// TwinCAT 3 PLC project SeedraPLC
// ProgramVersion: 3.1.4023.0
// libraries:
//   SPT Base Types, * (Beckhoff Automation LLC)
//   SPT Components, * (Beckhoff Automation LLC)
//   SPT Event Logger, * (Beckhoff Automation LLC)
//   SPT Motion Control, * (Beckhoff Automation LLC)
//   SPT Utilities, * (Beckhoff Automation LLC)
//   Tc2_EtherCAT, * (Beckhoff Automation GmbH)
//   Tc2_MC2, * (Beckhoff Automation GmbH)
//   Tc2_Standard, * (Beckhoff Automation GmbH)
//   Tc2_System, * (Beckhoff Automation GmbH)
//   Tc3_EventLogger, * (Beckhoff Automation GmbH)
//   Tc3_Module, * (Beckhoff Automation GmbH)
//   Tc3_PackML_V2, * (Beckhoff Automation GmbH)
//   VisuDialogs, * (System)
//   VisuSymbols,newest,System
// project tree:
//   / GlobalTextList.TcGTLO, MAIN.TcPOU, TaskPLC.TcTTO, VisualizationManager.TcVMO (not stored)
//   GVL/ IO.TcGVL, SafetyGlobalVariableList.TcGVL
//   Machine/Components/ FB_GantryXYCylinder.TcPOU, I_Cylinder.TcIO (not stored), ST_CylinderX_Command.TcDUT, ST_CylinderX_Config.TcDUT, ST_CylinderX_HMI.TcDUT, ST_CylinderX_Status.TcDUT
//   Machine/ FB_GantryXYZ.TcPOU, FB_Machine.TcPOU
//   Machine/VISUs/ V_MachineModule.TcVIS, V_Main.TcVIS, V_Module.TcVIS
// real-time tasks:
//   TASK TaskPLC: cycle T#10ms, priority 20, ADS port 350
// motion (NC):
//   TASK NC-Task 1 SAF: cycle T#2ms, priority 4, ADS port 501
//   TASK NC-Task 1 SVB: cycle T#10ms, priority 8, ADS port 511
//   AXIS AxisX (id 1)
//     PositionAreaControl: Enable=false
//     TargetPosControl: Enable=false
//     OtherSettings: AllowMotionCmdToSlave=true
//     encoder EncType=1
//     drive DrvType=5
//       Analog: TorqueSetpointScale=10, ScaleFactorActTorque=0.1
//       TimeComp: TaskDelayCycles=1
//     controller CtrType=1
//       CtrPara: PriorControlFactor=1
//         PosDiffControl: Enable=false
//         Observer: BandWidth=20
//   AXIS AxisY (id 2)
//     PositionAreaControl: Enable=false
//     TargetPosControl: Enable=false
//     OtherSettings: AllowMotionCmdToSlave=true
//     encoder EncType=1
//     drive DrvType=5
//       Analog: TorqueSetpointScale=10, ScaleFactorActTorque=0.1
//       TimeComp: TaskDelayCycles=1
//     controller CtrType=1
//       CtrPara: PriorControlFactor=1
//         PosDiffControl: Enable=false
//         Observer: BandWidth=20
//   AXIS AxisZ (id 3)
//     PositionAreaControl: Enable=false
//     TargetPosControl: Enable=false
//     OtherSettings: AllowMotionCmdToSlave=true
//     encoder EncType=1
//     drive DrvType=5
//       Analog: TorqueSetpointScale=10, ScaleFactorActTorque=0.1
//       TimeComp: TaskDelayCycles=1
//     controller CtrType=1
//       CtrPara: PriorControlFactor=1
//         PosDiffControl: Enable=false
//         Observer: BandWidth=20
// variable links:
//   SeedraPLC/SeedraPLC Instance <-> NC-Task 1 SAF/Axes/AxisX
//     TaskPLC Inputs/MAIN.Seedra.GantryXYZ.AxisX.BasicAxis._Axis.NcToPlc <-> Outputs/ToPlc
//     TaskPLC Outputs/MAIN.Seedra.GantryXYZ.AxisX.BasicAxis._Axis.PlcToNc <-> Inputs/FromPlc
//   SeedraPLC/SeedraPLC Instance <-> NC-Task 1 SAF/Axes/AxisY
//     TaskPLC Inputs/MAIN.Seedra.GantryXYZ.AxisY.BasicAxis._Axis.NcToPlc <-> Outputs/ToPlc
//     TaskPLC Outputs/MAIN.Seedra.GantryXYZ.AxisY.BasicAxis._Axis.PlcToNc <-> Inputs/FromPlc
//   SeedraPLC/SeedraPLC Instance <-> NC-Task 1 SAF/Axes/AxisZ
//     TaskPLC Inputs/MAIN.Seedra.GantryXYZ.AxisZ.BasicAxis._Axis.NcToPlc <-> Outputs/ToPlc
//     TaskPLC Outputs/MAIN.Seedra.GantryXYZ.AxisZ.BasicAxis._Axis.PlcToNc <-> Inputs/FromPlc

CONFIGURATION SeedraPLC
    RESOURCE PLC ON TwinCAT3
        TASK TaskPLC(INTERVAL := T#10ms, PRIORITY := 20);
        PROGRAM MAIN WITH TaskPLC : MAIN;
    END_RESOURCE
END_CONFIGURATION

// ---- Machine/Components/ST_CylinderX_Command.TcDUT
TYPE ST_CylinderX_Command :
    STRUCT
        RetractExtend  : BOOL;
        RetractCylinder : BOOL;
    END_STRUCT
END_TYPE

// ---- Machine/Components/ST_CylinderX_Config.TcDUT
TYPE ST_CylinderX_Config :
    STRUCT
        ExtendTime  : LREAL;
        RetractTime : LREAL;
    END_STRUCT
END_TYPE

// ---- Machine/Components/ST_CylinderX_HMI.TcDUT
TYPE ST_CylinderX_HMI :
    STRUCT
        Config  : ST_Cylinder_Config;
        Command : ST_CylinderX_Command;
        Status  : ST_CylinderX_Status;
    END_STRUCT
END_TYPE

// ---- Machine/Components/ST_CylinderX_Status.TcDUT
TYPE ST_CylinderX_Status :
    STRUCT
        Extended   : BOOL;
        Retracted  : BOOL;
        Extending  : BOOL;
        Retracting : BOOL;
    END_STRUCT
END_TYPE

// ---- GVL/IO.TcGVL
VAR_GLOBAL

	ProximitySensorX			AT%I*		:	BOOL;
	ProximitySensorY			AT%I*		:	BOOL;
	ProximitySensorZ			AT%I*		:	BOOL;
	kot : UDINT;


END_VAR

// ---- GVL/SafetyGlobalVariableList.TcGVL
{attribute 'qualified_only'}

VAR_GLOBAL
	
	eStop						 :BOOL;

(*	//State
	SafetySate: INT;
	ERR_ACK_RESETED : BOOL;
	AX5805_ErrACK_RESETED : BOOL;
	
	//TWinSafe Group
	ERR_FB						AT %I* :BOOL;
	ERR_COM						AT %I* :BOOL;
	ERR_OTHER					AT %I* :BOOL;
	IN_RUN						AT %I* :BOOL;
	RUN_STOP					AT %Q* :BOOL;
	ERR_ACK						AT %Q* :BOOL;
	
	//AX580x
	AX5805_Error_Ch1			AT %I* :BOOL;
	AX5805_Error_Ch2			AT %I* :BOOL;
	AX5805_STO_State_Ch1		AT %I* :BOOL;
	AX5805_STO_State_Ch2		AT %I* :BOOL;
	AX5805_ErrACK				AT %Q* :BOOL;
	
	//Other
	SAFETY_Permission			AT %I* :BOOL;
	RestartFBs_TSG				AT %Q* :BOOL;
*)

END_VAR

// ---- MAIN.TcPOU
PROGRAM MAIN

	VAR
		Seedra          : FB_Machine := (Name := 'SeedraMAIN');
		InitComplete    : BOOL;
	END_VAR

CyclicLogic();

METHOD CyclicLogic
VAR_INPUT
END_VAR
IF NOT InitComplete THEN
    InitComplete := Initialize();
    RETURN;
END_IF

//Machine support HMI & Production Monitor


//Machine Cyclic Logic
Seedra.CyclicLogic();
END_METHOD

METHOD Initialize : BOOL
VAR_INPUT
END_VAR
//Top level machine initialization should happen here, in the main initialization method. Each subsequent "layer" of modules will be named within their respective "parent" intialize method
_AppInfo.KeepOutputsOnBP := TRUE;
Initialize := TRUE;
END_METHOD

END_PROGRAM

// ---- Machine/FB_Machine.TcPOU
FUNCTION_BLOCK FB_Machine EXTENDS FB_PackML_BaseModule // IMPLEMENTS I_ControlsProductionRate
VAR
    // Sub Modules
    GantryXYZ   : FB_GantryXYZ  := (Name := 'Gantry', LogStateChanges := TRUE);

    //Initial List of Components
    ipComponents_Init : ARRAY[1..Parameters_PackML_Base.MAX_NO_OF_COMPONENTS] OF I_ComponentBase := [];

	//Alarms for this module
	MachineAlarms : ARRAY[1..MACHINE_ALARM_COUNT] OF FB_TcAlarm;

END_VAR

VAR CONSTANT
    MACHINE_ALARM_COUNT : INT := 6;
END_VAR


METHOD PROTECTED Clearing
VAR
	i				: UDINT;
	SubModulesReady : BOOL := TRUE;
END_VAR
CASE SequenceState OF
    0:
        NoStateTasksToComplete := FALSE;
        SequenceState          := SequenceState + 10;
    10:
        
       	MachineAlarms[E_Seedra.EmergencyStop].Clear(0, 0);
        SequenceState := SequenceState + 10;
    20:
    	 StateTasksComplete := TRUE; 
END_CASE

SUPER^.Clearing();
END_METHOD

METHOD PROTECTED CreateEvents
VAR_INPUT
END_VAR
// Add your event creation here
F_CreateAllEventsInClass(Alarms     := MachineAlarms,
                         ClassSize  := SIZEOF(TC_Events.Seedra),
                         pInitEvent := ADR(TC_EVENTS.Seedra.InitReferenceEvent),
                         Prefix     := Name);
// Super call to base
SUPER^.CreateEvents();
END_METHOD

METHOD CyclicLogic
VAR_INPUT
END_VAR

IF NOT _InitComplete THEN
    _InitComplete := Initialize();
    RETURN;
END_IF

SUPER^.CyclicLogic();

//Here the alarms will raise and clear on its own if the input changes
IF SafetyGlobalVariableList.eStop AND NOT MachineAlarms[E_Seedra.EmergencyStop].bRaised THEN
	RaiseAlarmWithStrings(MachineAlarms[E_Seedra.EmergencyStop],'','');
	//ELSIF NOT SafetyGlobalVariableList.eStop THEN
		//MachineAlarms[E_Seedra.EmergencyStop].Clear(0, 0);
END_IF
END_METHOD

METHOD PROTECTED Execute
CASE _CurrentMode OF

	//=================================PRODUCTION MODE==================================
	E_PMLUnitMode.ePMLUnitMode_Production:
		CASE SequenceState OF
			0:
				NoStateTasksToComplete := FALSE;

				//Advance Gantry to Resetting (Homing)
				GantryXYZ.ChangeState(E_PMLCommand.ePMLCommand_Start);
				
				SequenceState := SequenceState + 10;
					
			10:
				StateTasksComplete := TRUE;
				StateComplete();
				
			
		END_CASE

	//=================================MAINTENANCE & MANUAL MODE==================================
	E_PMLUnitMode.ePMLUnitMode_Maintenance, E_PMLUnitMode.ePMLUnitMode_Manual:
		;
END_CASE
END_METHOD

//! @summary Provides interlocks for HMI control and updates HMI status information for this module
METHOD PROTECTED HMICommunication

//! @description This method is called cyclically by <c>CyclicLogic()</c>

IF SafetyGlobalVariableList.eStop THEN
	PackMLBaseModule_HMI.Status.Error := TRUE;
	THIS^._Error := TRUE;
END_IF



SUPER^.HMICommunication();
END_METHOD

METHOD PROTECTED HMIPermissions
//General Mode Based Monitoring and handling of HMI control
CASE _CurrentMode OF
   
 E_PMLUnitMode.ePMLUnitMode_Production:
        CASE _CurrentState OF
            E_PMLState.ePMLState_Stopped:
				AllowHMIControl(ThisModuleOnly := FALSE);
            E_PMLState.ePMLState_Idle:
				AllowHMIControl(ThisModuleOnly := FALSE);
            E_PMLState.ePMLState_Suspended:
         		AllowHMIControl(ThisModuleOnly := FALSE);
            E_PMLState.ePMLState_Execute:
            	AllowHMIControl(ThisModuleOnly := FALSE); 
            E_PMLState.ePMLState_Aborted:
                AllowHMIControl(ThisModuleOnly := FALSE); 
            E_PMLState.ePMLState_Held:
                AllowHMIControl(ThisModuleOnly := FALSE); 
            E_PMLState.ePMLState_Complete:
          		AllowHMIControl(ThisModuleOnly := FALSE); 
        END_CASE
		
    E_PMLUnitMode.ePMLUnitMode_Manual:
        AllowHMIControl(ThisModuleOnly := FALSE); 
	E_PMLUnitMode.ePMLUnitMode_Maintenance:
        AllowHMIControl(ThisModuleOnly := FALSE); 
END_CASE
END_METHOD

METHOD PROTECTED Initialize : BOOL
VAR
    i : UDINT; //Generic iteration value
END_VAR
Initialize := FALSE;
CASE DescendantSequenceState OF
    0:
		RegisterSubmodule(GantryXYZ);

        _LogModeChanges         := FALSE;
        _LogStateChanges        := FALSE;
  
	    DescendantSequenceState := DescendantSequenceState + 10;
    10:
        DescendantSequenceState := DescendantSequenceState + 10;
    20:
        //Copy Mode names
        FOR i := 1 TO 3 DO
            ModeNames[i] := F_UnitModeToString(UDINT_TO_DINT(i));
        END_FOR

        DescendantSequenceState := DescendantSequenceState + 10;
    30:
        // Initialize Recipes 

        DescendantSequenceState := DescendantSequenceState + 10;
    40:
        //Call the Super
        IF SUPER^.Initialize() THEN
            DescendantSequenceState := DescendantSequenceState + 10;
        END_IF
    50:
        Initialize := TRUE;
END_CASE
END_METHOD

METHOD PROTECTED Resetting
VAR
	i				: UDINT;
	SubModulesReady : BOOL := TRUE;
END_VAR
CASE _CurrentMode OF

	//=================================PRODUCTION MODE==================================
	E_PMLUnitMode.ePMLUnitMode_Production:
		CASE SequenceState OF
			0:
				NoStateTasksToComplete := FALSE;

				//Advance Gantry to Resetting (Homing)
				GantryXYZ.ChangeState(E_PMLCommand.ePMLCommand_Reset);
				
				SequenceState := SequenceState + 10;
					
			10:
				StateTasksComplete := TRUE;
				SUPER^.Resetting();
				
			
		END_CASE

	//=================================MAINTENANCE & MANUAL MODE==================================
	E_PMLUnitMode.ePMLUnitMode_Maintenance, E_PMLUnitMode.ePMLUnitMode_Manual:
		;
END_CASE
END_METHOD

//! @summary This method monitors <b>submodules</b> within this PackML module and initiates fault responses as required
METHOD PROTECTED SubModuleMonitor : BOOL
VAR
	AlarmResponses : ARRAY[0..4] OF E_AlarmResponse; //Temporary response array	
	i			   : UDINT;
END_VAR

//! @description This method is called cyclically by <c>CyclicLogic()</c>
// Check the sub Modules for Alarm Severity
SUPER^.SubModuleMonitor();

//Check the alarms at the machine level
_CurrentAlarmSeverity := F_GetMaxSeverityRaised(Alarms := MachineAlarms, CurrentSeverity := _CurrentAlarmSeverity);

//Check the severity of the machine level alarms
IF _CurrentState <> E_PMLState.ePMLState_Aborted AND _CurrentState <> E_PMLState.ePMLState_Aborting AND _CurrentState <> E_PMLState.ePMLState_Clearing AND
   _CurrentState <> E_PMLState.ePMLState_Stopped AND _CurrentState <> E_PMLState.ePMLState_Stopping THEN
    AlarmResponses := _ParentFaultResponseDefinitions;
    CASE AlarmResponses[CurrentAlarmSeverity] OF
        E_AlarmResponse.Abort_ImmediateError:
            AbortImmediateError(Name, TRUE);
			AbortImmediateError(Name, FALSE);
        E_AlarmResponse.Abort_Immediate:
            AbortImmediate();
        E_AlarmResponse.Stop_Immediate:
            StopImmediate();
        E_AlarmResponse.Stop_Controlled:
            StopControlled();
        E_AlarmResponse.Hold_Immediate:
            HoldImmediate();
        E_AlarmResponse.Suspend_Immediate:
            SuspendImmediate();
        E_AlarmResponse.Suspend_Controlled:
            SuspendControlled();
        E_AlarmResponse.NoResponse:
            ;
    END_CASE
ELSIF _CurrentState = E_PMLState.ePMLState_Stopped OR _CurrentState = E_PMLState.ePMLState_Stopping THEN
    AlarmResponses := _ParentFaultResponseDefinitions;
    CASE AlarmResponses[CurrentAlarmSeverity] OF
        E_AlarmResponse.Abort_ImmediateError:
            AbortImmediateError(Name, TRUE);
        E_AlarmResponse.Abort_Immediate:
            AbortImmediate();
        E_AlarmResponse.NoResponse:
            ;
    END_CASE
END_IF
END_METHOD

END_FUNCTION_BLOCK

// ---- Machine/FB_GantryXYZ.TcPOU
FUNCTION_BLOCK FB_GantryXYZ EXTENDS FB_PackML_BaseModule 
VAR
    // Sub module definitions here

    // List of sub modules
    ipSubModules_Init : ARRAY[1..Parameters_PackML_Base.MAX_NO_OF_SUBMODULES] OF I_PackML_BaseModule := [];

    // Component definitions here
    AxisX       		: FB_Component_BasicAxis 		:= (Name := 'AxisX');
    AxisY    			: FB_Component_BasicAxis 		:= (Name := 'AxisY');
	AxisZ				: FB_Component_BasicAxis		:= (Name := 'AxisZ');
    GantryCylinder		: FB_GantryXYCylinder			:= (Name := 'Cylinder');

    //Alarms for this module
    GantryAlarms : ARRAY[1..GANTRY_ALARM_COUNT] OF FB_TcAlarm;

	//IO
	LimitSwitchX :BOOL;
	LimitSwitchY :BOOL;
	LimitSwitchZ :BOOL;

	HomeComplete :BOOL;
	


END_VAR

VAR CONSTANT
    GANTRY_ALARM_COUNT : INT := 5;
END_VAR

METHOD PROTECTED Clearing
VAR
	i				: UDINT;
	SubModulesReady : BOOL := TRUE;
END_VAR
CASE SequenceState OF
    0:
        NoStateTasksToComplete := FALSE;
        SequenceState          := SequenceState + 10;
    10:
        //Reset any alarms that get latched
        GantryAlarms[E_Gantry.StartTimeout].Clear(0, 0);
        SequenceState := SequenceState + 10;
    20:
        // Enable here
        AxisX.Enable();
        AxisY.Enable();
		AxisZ.Enable();

        // Check enabled here
        IF AxisX.Enabled AND AxisY.Enabled AND AxisZ.Enabled THEN
            SequenceState := SequenceState + 10;
        END_IF
    30:
        StateTasksComplete := TRUE;
END_CASE

SUPER^.Clearing();
END_METHOD

METHOD PROTECTED CreateEvents
VAR_INPUT
END_VAR
// Add your event creation here
F_CreateAllEventsInClass(Alarms     := GantryAlarms,
                         ClassSize  := SIZEOF(TC_EVENTS.Gantry),
                         pInitEvent := ADR(TC_EVENTS.Gantry.InitReferenceEvent),
                         Prefix     := _Name);

// Super call to base
SUPER^.CreateEvents();
END_METHOD

METHOD CuttingBoxFiveSides : BOOL

VAR_INST
	Step : INT ;	
END_VAR



(*
	F			H
	|			|
D---+-----------+---C
	|			|
	|			| 
B---+-----------+---A
	|			|
	E			G
*)
	CASE Step OF
		
		0:  

//Print Info
			
			Trace('Start Cutting Box Five Sides');
			
			Step := Step + 10;	

		10:	//Set Speed

//			AxisX.Velocity := 10; 
//			AxisY.Velocity := 10;
//			AxisZ.Velocity := 5;
			
			Step := Step + 160;

//		20:	//Positioning Motion to A
   			
//			AxisX.MoveAbsolute(0,0);
//			AxisY.MoveAbsolute(250,0);		
			
//			Step := Step + 10; 
		
//		30: //Set Cutting Height
			
//			AxisZ.MoveAbsolute(-30,0);
			
//			Step := Step + 10;

//		40: //Cutting Motion from A to B
			
//			AxisX.MoveAbsolute(500,0);		
			
//			Step := Step + 10;
		
//		50: //Return from Cutting Height 
			
//			AxisZ.MoveAbsolute(50,0);

//			Step := Step + 10;
		
//		60: //Positioning Motion from B to C
			
//			AxisX.MoveAbsolute(0,0);
//			AxisY.MoveAbsolute(50,0);
	
//			Step := Step + 10;

//		70: //Set Cutting Height
		
//			AxisZ.MoveAbsolute(0,0);

//			Step := Step + 10;

//		80: //Cutting Motion from C to D
			
//			AxisX.MoveAbsolute(500,0);
//			AxisY.MoveAbsolute(50,0);

//			Step := Step + 10;

//		90: //Return from Cutting Height 
			
//			AxisZ.MoveAbsolute(50,0);
			
//			Step := Step + 10;

//		100: //Positioning Motion from D to E
			
//			AxisX.MoveAbsolute(450,0);
//			AxisY.MoveAbsolute(300,0);

//			Step := Step + 10;
		
//		110: //Set Cutting Height 	
			
//			AxisZ.MoveAbsolute(0,0);
	
//			Step := Step + 10;

//		120: //Cutting Motion from E to F

//			AxisX.MoveAbsolute(450,0);
//			AxisY.MoveAbsolute(0,0);
			
//			Step := Step + 10;

//		130: //Return from Cutting Height 

//			AxisZ.MoveAbsolute(50,0);
			
//			Step := Step + 10;

//		140: //Positioning Motion from F to G

//			AxisX.MoveAbsolute(50,0);
//			AxisY.MoveAbsolute(300,0);

//			Step := Step + 10;

//		150: //Cutting Motion from G to H
  
//			AxisX.MoveAbsolute(50,0);
//			AxisY.MoveAbsolute(0,0);

//			Step := Step + 10;

//		160: //Return from Cutting Height 
	
//			AxisZ.MoveAbsolute(50,0);

//			Step := Step + 10;

		170: 

//Return to ZERO
////			AxisX.MoveAbsolute(0,0);
//			AxisY.MoveAbsolute(0,0);
			CuttingBoxFiveSides := TRUE;
			Step := 0;
			Trace('Box Five Sides is Cut');
		
			

		

			
	END_CASE
END_METHOD

METHOD CyclicLogic
VAR_INPUT
END_VAR
IF NOT _InitComplete THEN
    _InitComplete := Initialize();
    RETURN;
END_IF

SUPER^.CyclicLogic();

//Set the current alarm severity for this module
_CurrentAlarmSeverity := F_GetMaxSeverityRaised(Alarms := GantryAlarms, CurrentSeverity := _CurrentAlarmSeverity);

//Simulate Alarm Messaging
END_METHOD

METHOD PROTECTED Execute
CASE _CurrentMode OF

	//=================================PRODUCTION MODE==================================
	E_PMLUnitMode.ePMLUnitMode_Production:
		CASE SequenceState OF
			0:
				NoStateTasksToComplete := FALSE;
				
				IF NOT CuttingBoxFiveSides() THEN
					CuttingBoxFiveSides();	
				ELSE
					SequenceState := SequenceState + 10;
				END_IF		
				
			10:		
				StateTasksComplete := TRUE;
				StateComplete();
			END_CASE

	//=================================MAINTENANCE & MANUAL MODE==================================
	E_PMLUnitMode.ePMLUnitMode_Maintenance, E_PMLUnitMode.ePMLUnitMode_Manual:
		;
END_CASE
END_METHOD

METHOD PROTECTED HMIPermissions
//General Mode Based Monitoring and handling of HMI control
CASE _CurrentMode OF
   
 E_PMLUnitMode.ePMLUnitMode_Production:
        CASE _CurrentState OF
            E_PMLState.ePMLState_Stopped:
				AllowHMIControl(ThisModuleOnly := FALSE);
            E_PMLState.ePMLState_Idle:
				AllowHMIControl(ThisModuleOnly := FALSE);
            E_PMLState.ePMLState_Suspended:
         		AllowHMIControl(ThisModuleOnly := FALSE);
            E_PMLState.ePMLState_Execute:
            	AllowHMIControl(ThisModuleOnly := FALSE); 
            E_PMLState.ePMLState_Aborted:
                AllowHMIControl(ThisModuleOnly := FALSE); 
            E_PMLState.ePMLState_Held:
                AllowHMIControl(ThisModuleOnly := FALSE); 
            E_PMLState.ePMLState_Complete:
          		AllowHMIControl(ThisModuleOnly := FALSE); 
        END_CASE
		
    E_PMLUnitMode.ePMLUnitMode_Manual:
        AllowHMIControl(ThisModuleOnly := FALSE); 
	E_PMLUnitMode.ePMLUnitMode_Maintenance:
        AllowHMIControl(ThisModuleOnly := FALSE); 
END_CASE
END_METHOD

METHOD Homing : BOOL

VAR_INST
	Step : INT ;	
END_VAR
	CASE Step OF
		
		0: 
			Trace('Home X');
			AxisX.Home();
			Step := Step + 10; 
		10:
			Trace('Home Y');
			AxisY.Home();
			Step := Step + 10;
	
		20:	
			Trace('Home Z');
			AxisZ.Home();
			Homing := TRUE;
			Step := 0;	

	END_CASE
END_METHOD

//! @summary Basic module initialization logic
METHOD PROTECTED Initialize : BOOL;
VAR
    i                        : UDINT;
    varInfo                  : __SYSTEM.VAR_INFO;
    AllSubUnitsInitialized   : BOOL := TRUE;
    AllComponentsInitialized : BOOL := TRUE;
END_VAR

//! @description This method is called by <c>CyclicLogic()</c> as required
Initialize := FALSE;
CASE DescendantSequenceState OF
    0:
		RegisterComponent(AxisX);
		RegisterComponent(AxisY);	
		RegisterComponent(AxisZ);	
		RegisterComponent(GantryCylinder);
		
        _LogModeChanges         := FALSE;
        _LogStateChanges        := FALSE;
        DescendantSequenceState := DescendantSequenceState + 10;
    10:
        DescendantSequenceState := DescendantSequenceState + 10;
    20:
        //Copy Mode names
        FOR i := 1 TO 3 DO
            ModeNames[i] := F_UnitModeToString(UDINT_TO_DINT(i));
        END_FOR

        DescendantSequenceState := DescendantSequenceState + 10;
    30:
        //Call the Super
        IF SUPER^.Initialize() THEN
            DescendantSequenceState := DescendantSequenceState + 10;
        END_IF
    40:
        Initialize := TRUE;
END_CASE
END_METHOD

METHOD PROTECTED Resetting
VAR
	i				: UDINT;
	SubModulesReady : BOOL := TRUE;
END_VAR
CASE _CurrentMode OF

	//=================================PRODUCTION MODE==================================
	E_PMLUnitMode.ePMLUnitMode_Production:
		CASE SequenceState OF
			0:
				NoStateTasksToComplete := TRUE;
				
				IF NOT Homing() THEN
					Homing();
				ELSE
					SequenceState := SequenceState + 10;	
				END_IF		
				
			10:		
				StateTasksComplete := TRUE;
				SUPER^.Resetting();
		END_CASE

	//=================================MAINTENANCE & MANUAL MODE==================================
	E_PMLUnitMode.ePMLUnitMode_Maintenance, E_PMLUnitMode.ePMLUnitMode_Manual:
		;
END_CASE
END_METHOD

END_FUNCTION_BLOCK

// ---- Machine/Components/FB_GantryXYCylinder.TcPOU
(*	This FB is used for a single output solenoid 
	It uses the times to say when Extended/Retracted  	
	It starts assuming retracted and the output off.
*)
FUNCTION_BLOCK FB_GantryXYCylinder EXTENDS FB_ComponentBase IMPLEMENTS I_Cylinder
VAR
    //Output
    Output AT %Q* : BOOL;

    // Internal variables
    _ExtendRequest  : BOOL;
    _RetractRequest : BOOL;
    _Extended       : BOOL;
    _Retracted      : BOOL;
    _Extending      : BOOL;
    _Retracting     : BOOL;
    _ExtendTime     : LREAL := 1000; // Default time 1s
    _RetractTime    : LREAL := 1000; // Default time 1s

    // Timer for Extend/Retract
    Extend_TON    : TON;
    Retract_TON   : TON;
    Extend_RTRIG  : R_TRIG;
    Retract_RTRIG : R_TRIG;

    //HMI 
    Cylinder_HMI : ST_CylinderX_HMI;
END_VAR

METHOD PROTECTED CreateEvents
VAR_INPUT
END_VAR
SUPER^.CreateEvents();
END_METHOD

METHOD CyclicLogic
//One shot the requests
Extend_RTRIG(CLK := _ExtendRequest);
Retract_RTRIG(CLK := _RetractRequest);

//Handle Extend
IF Extend_RTRIG.Q THEN
    Output          := TRUE;
    _Extending      := TRUE;
    _Retracting     := FALSE;
    _Retracted      := FALSE;
    _RetractRequest := FALSE;
END_IF

//Handle Retract
IF Retract_RTRIG.Q THEN
    Output         := FALSE;
    _Extending     := FALSE;
    _Retracting    := TRUE;
    _Extended      := FALSE;
    _ExtendRequest := FALSE;
END_IF

//Handle the time to Extend/Retract
Extend_TON(IN := _Extending, PT := LREAL_TO_TIME(_ExtendTime));
Retract_TON(IN := _Retracting, PT := LREAL_TO_TIME(_RetractTime));
IF Extend_TON.Q THEN
    _Extended  := TRUE;
    _Extending := FALSE;
END_IF

IF Retract_TON.Q THEN
    _Retracted  := TRUE;
    _Retracting := FALSE;
END_IF

SUPER^.CyclicLogic();
END_METHOD

METHOD Extend
_ExtendRequest  := TRUE;
_RetractRequest := FALSE;
END_METHOD

PROPERTY Extended : BOOL
GET
Extended := _Extended;
END_GET
END_PROPERTY

PROPERTY ExtendTime : LREAL
GET
ExtendTime := _ExtendTime;
END_GET
SET
END_SET
END_PROPERTY

METHOD PROTECTED HMICommunication
VAR_INPUT
END_VAR
SUPER^.HMICommunication();

//Handle the requests to extend and retract
IF ComponentBase_HMI.Status.HMIControlAvailable THEN
    IF Cylinder_HMI.Command.RetractExtend THEN
        Extend();
    ELSIF Cylinder_HMI.Command.RetractCylinder THEN
        Retract();
    END_IF
END_IF

//Update HMI status info
Cylinder_HMI.Status.Extended    := _Extended;
Cylinder_HMI.Status.Extending   := _Extending;
Cylinder_HMI.Status.Retracted   := _Retracted;
Cylinder_HMI.Status.Retracting  := _Retracting;
Cylinder_HMI.Config.ExtendTime  := _ExtendTime;
Cylinder_HMI.Config.RetractTime := _RetractTime;
END_METHOD

//! @summary Basic component initialization logic
METHOD PROTECTED Initialize : BOOL;

//! @description This method is called by <c>CyclicLogic()</c> as required
//Set the cylinder to retracted
IF Output THEN
    _Extended  := TRUE;
    _Retracted := FALSE;
ELSE
    _Extended  := FALSE;
    _Retracted := TRUE;
END_IF

_Extending      := FALSE;
_ExtendRequest  := FALSE;
_Retracting     := FALSE;
_RetractRequest := FALSE;

//Call base class Initialize
Initialize := SUPER^.Initialize();
END_METHOD

METHOD PROTECTED Monitoring
VAR_INPUT
END_VAR
_Busy    := _Extending OR _Retracting;
_Error   := FALSE;
_ErrorID := 0;
SUPER^.Monitoring();
END_METHOD

METHOD Retract
_ExtendRequest  := FALSE;
_RetractRequest := TRUE;
END_METHOD

PROPERTY Retracted : BOOL
GET
Retracted := _Retracted;
END_GET
END_PROPERTY

PROPERTY RetractTime : LREAL
GET
RetractTime := _RetractTime;
END_GET
SET
_RetractTime := RetractTime;
END_SET
END_PROPERTY

END_FUNCTION_BLOCK

// ---- GlobalTextList.TcGTLO
TEXTLIST GlobalTextList
  685 = '%s'
  470 = '>'
  680 = 'Abort'
  347 = 'BB8'
  452 = 'Clear'
  424 = 'EStop'
  744 = 'Hold'
  46 = 'Maintenance'
  904 = 'Manual'
  929 = 'Production'
  181 = 'Reset'
  77 = 'Start'
  354 = 'START'
  516 = 'State: %s'
  828 = 'Stop'
  98 = 'STOP'
  806 = 'Suspend'
  197 = 'Unhold'
  832 = 'Unsuspend'
  500 = 'V'
  277 = '▶'
  821 = '▶\nStart'
  266 = '▶Start'
END_TEXTLIST

// ---- Machine/VISUs/V_MachineModule.TcVIS
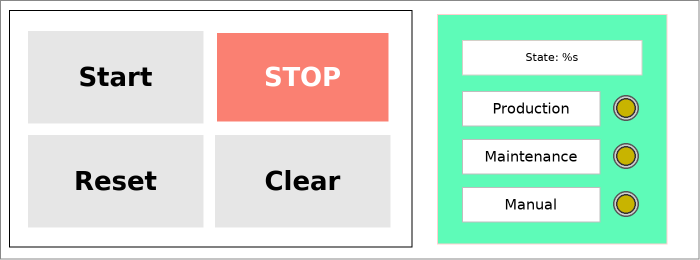
VISUALIZATION V_MachineModule  // 700x260
VAR_IN_OUT
	HMI : ST_PackMLBaseModule_HMI;
END_VAR
    Frame (432,10 240x240)
        shows V_Module(HMI := HMI)
    RoundedRectangle (9,10 403x237)
    RoundedRectangle (28,31 175x92), "Start"
        OnMouseClick: execute { HMI.Command.State := E_PMLCommand.ePMLCommand_Start; }
    RoundedRectangle (215,135 175x92), "Clear"
        OnMouseClick: execute { HMI.Command.State := E_PMLCommand.ePMLCommand_Clear; }
    RoundedRectangle (28,135 175x92), "Reset"
        OnMouseClick: execute { HMI.Command.State := E_PMLCommand.ePMLCommand_Reset; }
    RoundedRectangle (215,31 175x92), "STOP"
        toggle SafetyGlobalVariableList.eStop
        OnMouseClick: execute { HMI.Command.State := E_PMLCommand.ePMLCommand_Clear; }
END_VISUALIZATION

// ---- Machine/VISUs/V_Main.TcVIS
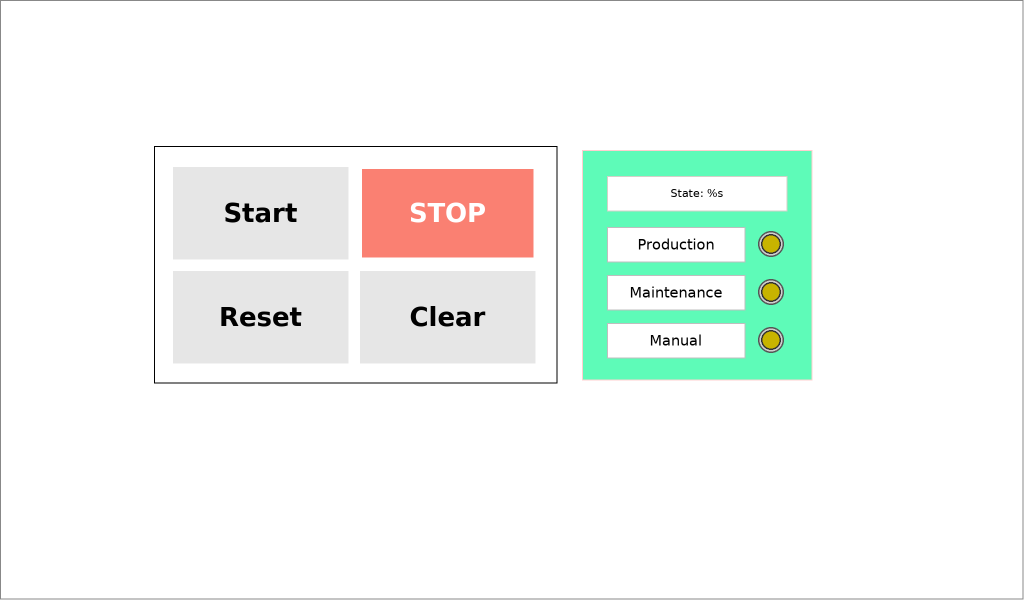
VISUALIZATION V_Main  // 1024x600
    Frame (145,136 700x260)
        shows V_MachineModule(HMI := MAIN.Seedra.PackMLBaseModule_HMI)
END_VISUALIZATION

// ---- Machine/VISUs/V_Module.TcVIS
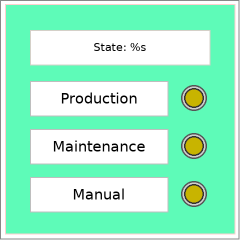
VISUALIZATION V_Module  // 240x240
VAR_IN_OUT
	HMI : ST_PackMLBaseModule_HMI;
END_VAR
    RoundedRectangle (5,4 230x230)
    Textfield (30,30 180x35), "State: %s", text variable: HMI.Status.State
    Lamp1 (179,83 30x30), variable: HMI.Status.Mode = E_PMLUnitMode.ePMLUnitMode_Production, style: Lamp-Lamp1-Yellow
    Lamp1 (179,131 30x30), variable: HMI.Status.Mode = E_PMLUnitMode.ePMLUnitMode_Maintenance, style: Lamp-Lamp1-Yellow
    Lamp1 (179,179 30x30), variable: HMI.Status.Mode = E_PMLUnitMode.ePMLUnitMode_Manual, style: Lamp-Lamp1-Yellow
    RoundedRectangle (30,81 138x35), "Production"
        OnMouseClick: execute { HMI.Command.Mode := E_PMLUnitMode.ePMLUnitMode_Production; }
    RoundedRectangle (30,129 138x35), "Maintenance"
        OnMouseClick: execute { HMI.Command.Mode := E_PMLUnitMode.ePMLUnitMode_Maintenance; }
    RoundedRectangle (30,177 138x35), "Manual"
        OnMouseClick: execute { HMI.Command.Mode := E_PMLUnitMode.ePMLUnitMode_Manual; }
END_VISUALIZATION
